INTERFACE I_MirrorCovers

METHOD AreCoversClosed : BOOL
VAR_INPUT
END_VAR
END_METHOD

METHOD AreCoversOpen : BOOL
VAR_INPUT
END_VAR
END_METHOD

METHOD CloseCover : BOOL
VAR_INPUT
	cover	: UINT;
END_VAR
END_METHOD

METHOD CloseCovers : BOOL
VAR_INPUT
END_VAR
END_METHOD

PROPERTY Error : BOOL
GET
END_GET
END_PROPERTY

METHOD IsCoverClosed : BOOL
VAR_INPUT
	cover	: UINT;	
END_VAR
END_METHOD

METHOD IsCoverOpen : BOOL
VAR_INPUT
	cover	: UINT;	
END_VAR
END_METHOD

METHOD OpenCover : BOOL
VAR_INPUT
	cover	: UINT;
END_VAR
END_METHOD

METHOD OpenCovers : BOOL
VAR_INPUT
END_VAR
END_METHOD

METHOD ResetCovers : BOOL
VAR_INPUT
END_VAR
END_METHOD

END_INTERFACE

(* stored: Version 1.1.0.1, ProductVersion 3.1.4026.8
   Itf I_MirrorCovers: Id {ce637c3e-ed3e-4174-8b7f-5e29873c1a6c}
   Method AreCoversClosed: Id {5bfd566b-f5d0-4c6f-9f10-d10c9709d33c}
   Method AreCoversOpen: Id {380f6690-4fbb-4ef1-9dc3-7a4959b63b35}
   Method CloseCover: Id {154de5be-ed9e-40a6-affb-5973b8c678f6}
   Method CloseCovers: Id {d170ed42-b733-4dca-b829-4ce12e150295}
   Property Error: Id {ff09ec7f-4b0d-4bfe-9bc0-a74f6b8e0c04}
   Get Get: Id {65d2e08e-b6f2-4c31-8697-8d42891b20d7}
   Method IsCoverClosed: Id {293aaa8b-84c3-44d0-8b88-9876c26d5402}
   Method IsCoverOpen: Id {7bf7d76e-c4ea-413e-8a66-508730888dbd}
   Method OpenCover: Id {a28ff9c8-eed2-49bd-83bd-d47b722e5119}
   Method OpenCovers: Id {47330435-4ab9-4214-8907-9d0910956eeb}
   Method ResetCovers: Id {8fd140fa-4504-401a-a6d2-edb6c92f8267} *)
